// Generic TCP/IP client: raw byte transport only, no protocol framing.
FUNCTION_BLOCK FB_TcpIpClient
VAR_INPUT
    bEnable             : BOOL;
    bReset              : BOOL;

    // Remote endpoint.
    Config              : stComm_UR_Config;

    // TRUE = continuously issue asynchronous receive requests.
    bReceiveEnable      : BOOL := TRUE;

    // Rising edge starts one send operation.
    bSend               : BOOL;
    pSendData           : PVOID;
    nSendSize           : UDINT;
END_VAR

VAR_OUTPUT
    // Connection status.
    bConnected          : BOOL;
    bReadyForSend       : BOOL;

    // Send status.
    bSendBusy           : BOOL;
    bSendDone           : BOOL;

    // Receive output. bRxNewData is a one-cycle pulse.
    bRxNewData          : BOOL;
    nRxBytes            : UDINT;
    aRxData             : ARRAY[0..2047] OF BYTE;

    // Error information.
    bError              : BOOL;
    nErrorId            : UDINT;
    sError              : STRING(80);
END_VAR

VAR
    // Beckhoff socket function blocks.
    fbSocketConnect     : FB_SocketConnect;
    fbSocketClose       : FB_SocketClose;
    fbSocketSend        : FB_SocketSend;
    fbSocketReceive     : FB_SocketReceive;
    fbReconnectDelay    : TON;

    hSocket             : T_HSOCKET;

    // Main state machine.
    nState              : USINT := 0;

    // Execute pulses for Beckhoff FBs.
    bConnectExecute     : BOOL;
    bCloseExecute       : BOOL;
    bSendExecute        : BOOL;
    bReceiveExecute     : BOOL;

    // Connection operation tracking.
    bConnectStarted     : BOOL;
    bCloseStarted       : BOOL;
    bReconnectAfterClose : BOOL;

    // Send operation tracking.
    bSendOld            : BOOL;
    bSendRise           : BOOL;
    bSendActive         : BOOL;
    bSendStarted        : BOOL;
    nActiveSendSize     : UDINT;
    aTxBuffer           : ARRAY[0..2047] OF BYTE;

    // Receive operation tracking.
    bReceiveActive      : BOOL;
    bReceiveStarted     : BOOL;
    nSocketRxBytes      : UDINT;
END_VAR

VAR CONSTANT
    C_STATE_DISCONNECTED    : USINT := 0;
    C_STATE_CONNECTING      : USINT := 10;
    C_STATE_CONNECTED       : USINT := 20;
    C_STATE_DISCONNECTING   : USINT := 30;
    C_STATE_ERROR_WAIT      : USINT := 90;

    C_BUFFER_SIZE           : UDINT := 2048;
END_VAR

// The socket FBs are called first: the execute flags set below are seen next cycle.
fbSocketConnect(
    sSrvNetId   := '',
    sRemoteHost := Config.sIpAddress,
    nRemotePort := UINT_TO_UDINT(Config.nPort),
    tTimeout    := Config.tTimeout,
    bExecute    := bConnectExecute,
    hSocket     => hSocket
);

fbSocketClose(
    sSrvNetId   := '',
    tTimeout    := Config.tTimeout,
    hSocket     := hSocket,
    bExecute    := bCloseExecute
);

fbSocketSend(
    sSrvNetId   := '',
    tTimeout    := Config.tTimeout,
    hSocket     := hSocket,
    bExecute    := bSendExecute,
    cbLen       := nActiveSendSize,
    pSrc        := ADR(aTxBuffer)
);

fbSocketReceive(
    sSrvNetId   := '',
    tTimeout    := Config.tTimeout,
    hSocket     := hSocket,
    bExecute    := bReceiveExecute,
    cbLen       := SIZEOF(aRxData),
    pDest       := ADR(aRxData),
    nRecBytes   => nSocketRxBytes
);

fbReconnectDelay(
    IN := (nState = C_STATE_ERROR_WAIT) AND bEnable,
    PT := T#1S
);


bConnectExecute := FALSE;
bCloseExecute := FALSE;
bSendExecute := FALSE;
bReceiveExecute := FALSE;

bSendDone := FALSE;
bRxNewData := FALSE;
nRxBytes := 0;

bSendRise := bSend AND NOT bSendOld;
bSendOld := bSend;

IF bReset THEN
    bError := FALSE;
    nErrorId := 0;
    sError := '';

    IF nState = C_STATE_ERROR_WAIT THEN
        nState := C_STATE_DISCONNECTED;
    END_IF
END_IF


CASE nState OF

    C_STATE_DISCONNECTED:
        bSendActive := FALSE;
        bSendStarted := FALSE;
        bReceiveActive := FALSE;
        bReceiveStarted := FALSE;
        bConnectStarted := FALSE;
        bCloseStarted := FALSE;

        IF bEnable THEN
            bConnectExecute := TRUE;
            nState := C_STATE_CONNECTING;
        END_IF


    C_STATE_CONNECTING:
        IF NOT bEnable THEN
            nState := C_STATE_DISCONNECTED;

        ELSE
            IF fbSocketConnect.bBusy THEN
                bConnectStarted := TRUE;
            END_IF

            IF fbSocketConnect.bError THEN
                bError := TRUE;
                nErrorId := fbSocketConnect.nErrId;
                sError := 'TCP connect error';

                bReconnectAfterClose := FALSE;
                nState := C_STATE_ERROR_WAIT;

            ELSIF bConnectStarted AND NOT fbSocketConnect.bBusy THEN
                bConnectStarted := FALSE;
                bError := FALSE;
                nErrorId := 0;
                sError := '';
                nState := C_STATE_CONNECTED;
            END_IF
        END_IF


    C_STATE_CONNECTED:
        IF NOT bEnable THEN
            bReconnectAfterClose := FALSE;
            bCloseStarted := FALSE;
            bCloseExecute := TRUE;
            nState := C_STATE_DISCONNECTING;

        ELSE

            IF bSendActive THEN

                IF fbSocketSend.bBusy THEN
                    bSendStarted := TRUE;
                END_IF

                IF fbSocketSend.bError THEN
                    bSendActive := FALSE;
                    bSendStarted := FALSE;

                    bError := TRUE;
                    nErrorId := fbSocketSend.nErrId;
                    sError := 'TCP send error';

                    bReconnectAfterClose := TRUE;
                    bCloseStarted := FALSE;
                    bCloseExecute := TRUE;
                    nState := C_STATE_DISCONNECTING;

                ELSIF bSendStarted AND NOT fbSocketSend.bBusy THEN
                    bSendActive := FALSE;
                    bSendStarted := FALSE;
                    bSendDone := TRUE;
                END_IF

            ELSIF bSendRise THEN

                IF (nSendSize = 0) OR (nSendSize > C_BUFFER_SIZE) OR (pSendData = 0) THEN
                    bError := TRUE;
                    nErrorId := 16#F002;
                    sError := 'Invalid TCP send buffer';

                ELSE
                    MEMCPY(destAddr := ADR(aTxBuffer), srcAddr := pSendData, n := nSendSize);

                    nActiveSendSize := nSendSize;
                    bSendActive := TRUE;
                    bSendStarted := FALSE;
                    bSendExecute := TRUE;
                END_IF
            END_IF


            IF bReceiveActive THEN

                IF fbSocketReceive.bBusy THEN
                    bReceiveStarted := TRUE;
                END_IF

                IF fbSocketReceive.bError THEN
                    bReceiveActive := FALSE;
                    bReceiveStarted := FALSE;

                    bError := TRUE;
                    nErrorId := fbSocketReceive.nErrId;
                    sError := 'TCP receive error';

                    bReconnectAfterClose := TRUE;
                    bCloseStarted := FALSE;
                    bCloseExecute := TRUE;
                    nState := C_STATE_DISCONNECTING;

                ELSIF bReceiveStarted AND NOT fbSocketReceive.bBusy THEN
                    bReceiveActive := FALSE;
                    bReceiveStarted := FALSE;

                    IF nSocketRxBytes > 0 THEN
                        nRxBytes := nSocketRxBytes;
                        bRxNewData := TRUE;
                    END_IF
                END_IF

            ELSIF bReceiveEnable THEN
                nSocketRxBytes := 0;
                bReceiveActive := TRUE;
                bReceiveStarted := FALSE;
                bReceiveExecute := TRUE;
            END_IF

        END_IF


    C_STATE_DISCONNECTING:
        IF fbSocketClose.bBusy THEN
            bCloseStarted := TRUE;
        END_IF

        IF fbSocketClose.bError THEN
            bCloseStarted := FALSE;

            IF bReconnectAfterClose AND bEnable THEN
                nState := C_STATE_ERROR_WAIT;
            ELSE
                bError := TRUE;
                nErrorId := fbSocketClose.nErrId;
                sError := 'TCP close error';
                nState := C_STATE_DISCONNECTED;
            END_IF

        ELSIF bCloseStarted AND NOT fbSocketClose.bBusy THEN
            bCloseStarted := FALSE;

            IF bReconnectAfterClose AND bEnable THEN
                nState := C_STATE_ERROR_WAIT;
            ELSE
                nState := C_STATE_DISCONNECTED;
            END_IF
        END_IF


    C_STATE_ERROR_WAIT:
        bSendActive := FALSE;
        bSendStarted := FALSE;
        bReceiveActive := FALSE;
        bReceiveStarted := FALSE;

        IF NOT bEnable THEN
            bError := FALSE;
            nErrorId := 0;
            sError := '';
            nState := C_STATE_DISCONNECTED;

        ELSIF bReset OR (Config.bAutoReconnect AND fbReconnectDelay.Q) THEN
            // Keep the previous error visible during the delay, then retry.
            bError := FALSE;
            nErrorId := 0;
            sError := '';
            nState := C_STATE_DISCONNECTED;
        END_IF


    ELSE
        bError := TRUE;
        nErrorId := 16#F0FF;
        sError := 'Invalid TCP state';
        nState := C_STATE_ERROR_WAIT;

END_CASE


bConnected := (nState = C_STATE_CONNECTED);
bSendBusy := bSendActive OR fbSocketSend.bBusy;
bReadyForSend := bConnected AND NOT bSendBusy AND NOT bError;

END_FUNCTION_BLOCK

(* stored: Version 1.1.0.1, ProductVersion 3.1.4026.18
   POU FB_TcpIpClient: Id {dbe0809b-56ae-4dcb-bda5-390ce8598918}, SpecialFunc None *)
